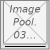
VISUALIZATION F_MainMenu_03  // 50x50
VAR_IN_OUT
	stMenuButton	: ST_HMIEButton_HMI;
END_VAR
    Image (3,0 44x44), invisible if: not stMenuButton.bVisible, image: ImagePool.03_Events
        OnMouseDown: execute { stMenuButton.bPushed := TRUE; }
    Line (5,46) (45,46), invisible if: not stMenuButton.bVisible or not stMenuButton.bActive, input disabled if: not stMenuButton.bEnable
END_VISUALIZATION

(* stored: Version 1.1.0.1
   Visu F_MainMenu_03: Id {9e2364bd-1f09-0803-12e6-98191ad6eef3} *)
